(* IEC 61131-3 sources: teller/JD_Teller_LC2_V11/Class/Timeconvert, 1 file *)

(* ---- Timeconvert.st ---- *)
(*!
<Class
	Name               = "Timeconvert"
	Revision           = "0.0"
	RealtimeTask       = "false"
	CyclicTask         = "false"
	BackgroundTask     = "true"
	DefBackground      = "100 ms"
	Sigmatek           = "false"
	OSInterface        = "false"
	HighPriority       = "false"
	Automatic          = "false"
	UpdateMode         = "Prescan"
	SharedCommandTable = "true"
	Objectsize         = "(284,120)">
	<Channels>
		<Server Name="ClassSvr" Visualized="false" Initialize="false" WriteProtected="true" Retentive="false"/>
		<Server Name="Tijd" Visualized="true" Initialize="false" WriteProtected="false" Retentive="false"/>
		<Client Name="Milisecs" Required="true" Internal="false"/>
	</Channels>
</Class>
*)
Timeconvert : CLASS
  //Servers:
	ClassSvr 	: SvrChCmd_DINT;
	Tijd 	: SvrCh_DINT;
  //Clients:
	Milisecs 	: CltCh_DINT;
  //Variables:
  //Functions:

	FUNCTION VIRTUAL GLOBAL Init;

	FUNCTION VIRTUAL GLOBAL Background
		VAR_INPUT
			EAX 	: UDINT;
		END_VAR
		VAR_OUTPUT
			state (EAX) 	: UDINT;
		END_VAR;

	FUNCTION VIRTUAL GLOBAL Tijd::Read
		VAR_OUTPUT
			output (EAX) 	: DINT;
		END_VAR;

	FUNCTION VIRTUAL GLOBAL Tijd::Write
		VAR_INPUT
			input (EAX) 	: DINT;
		END_VAR
		VAR_OUTPUT
			result (EAX) 	: DINT;
		END_VAR;
  //Tables:
	FUNCTION @STD
		VAR_OUTPUT
			ret_code	: CONFSTATES;
		END_VAR;
	FUNCTION GLOBAL TAB @CT_;
END_CLASS;

FUNCTION VIRTUAL GLOBAL Timeconvert::Init

Tijd := 2;

END_FUNCTION

FUNCTION VIRTUAL GLOBAL Timeconvert::Background
	VAR_INPUT
		EAX 	: UDINT;
	END_VAR
	VAR_OUTPUT
		state (EAX) 	: UDINT;
	END_VAR

  Milisecs := Milisecs.Read();
  Tijd := Milisecs/60000;

	state := READY;

END_FUNCTION

FUNCTION VIRTUAL GLOBAL Timeconvert::Tijd::Read
	VAR_OUTPUT
		output (EAX) 	: DINT;
	END_VAR

  Tijd := Milisecs/60000;
	output := Tijd;

END_FUNCTION

FUNCTION VIRTUAL GLOBAL Timeconvert::Tijd::Write
	VAR_INPUT
		input (EAX) 	: DINT;
	END_VAR
	VAR_OUTPUT
		result (EAX) 	: DINT;
	END_VAR

	Tijd := input;
  Milisecs := Tijd*60000;
  Milisecs.Write (Milisecs);
 	result := Tijd;

END_FUNCTION
